# EPICS substitutions: iocBoot/iocGamryTest/Gamry.substitutions
file "$(GAMRY)/GamryApp/Db/Interface1010E.template"
{
pattern
{    P,        PORT,       ADDR}
{   Gamry,   Gamry_1,     0}
}
